{attribute 'qualified_only'}
TYPE E_PackMLCommand :
(
	None		:= 0,
	Reset		:= 1,
	Start		:= 2,
	Stop		:= 3,
	Hold		:= 4,
	Unhold		:= 5,
	Suspend		:= 6,
	Unsuspend	:= 7,
	Abort		:= 8,
	Clear		:= 9
);
END_TYPE

(* stored: Version 1.1.0.1, ProductVersion 3.1.4026.18
   DUT E_PackMLCommand: Id {41dcc4de-90f2-4d77-94c8-7b4e3ff94f76} *)
